TYPE ST_MachineState :
STRUCT

	bStartup	 : BOOL;		
	bStartupDone : BOOL;
	bAborting 	 : BOOL;
	bResetting	 : BOOL;
	bStarting	 : BOOL;
	bRunning	 : BOOL;

END_STRUCT
END_TYPE

(* stored: Version 1.1.0.1, ProductVersion 3.1.4024.9
   DUT ST_MachineState: Id {b794778f-ca53-4e7f-87bb-35c4e79dd035} *)
